# B&R Automation Studio project DuctLines (part 7)

#### Cyclic.ld
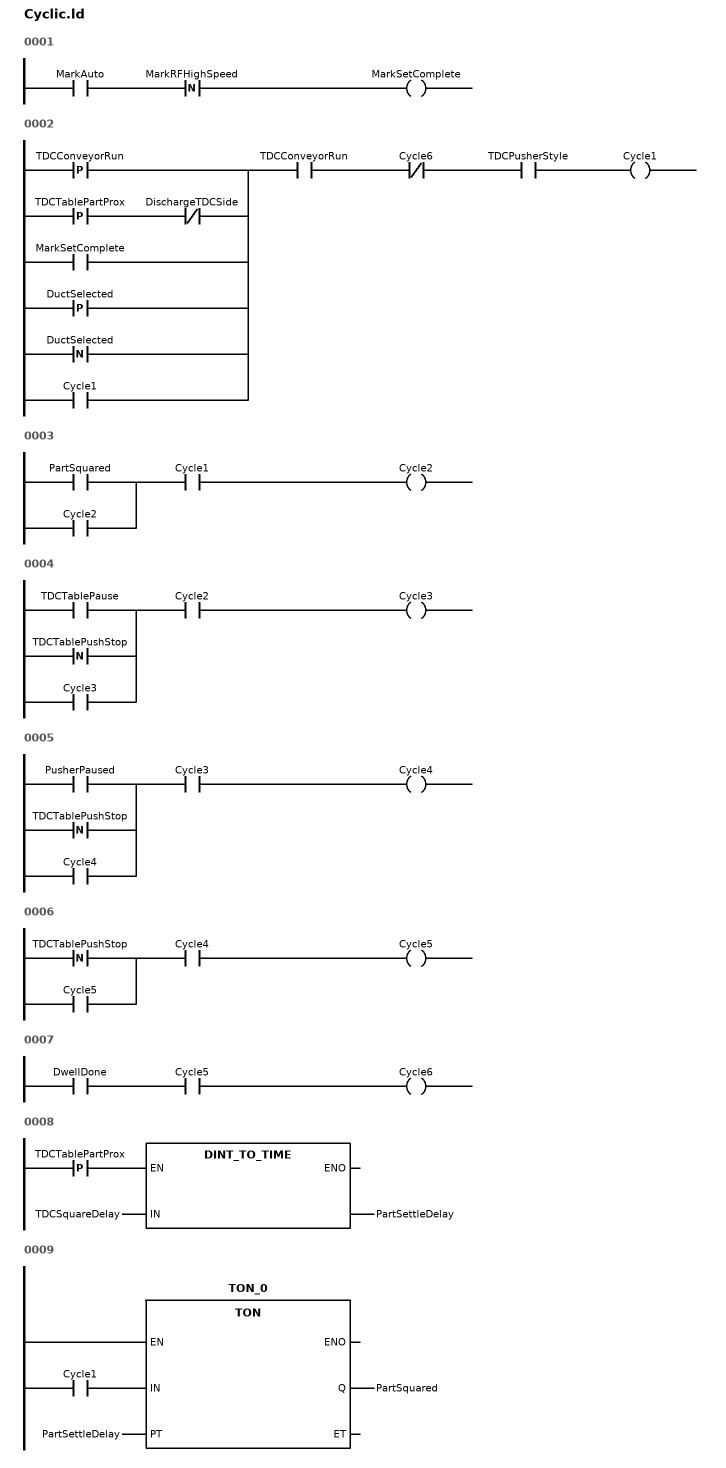
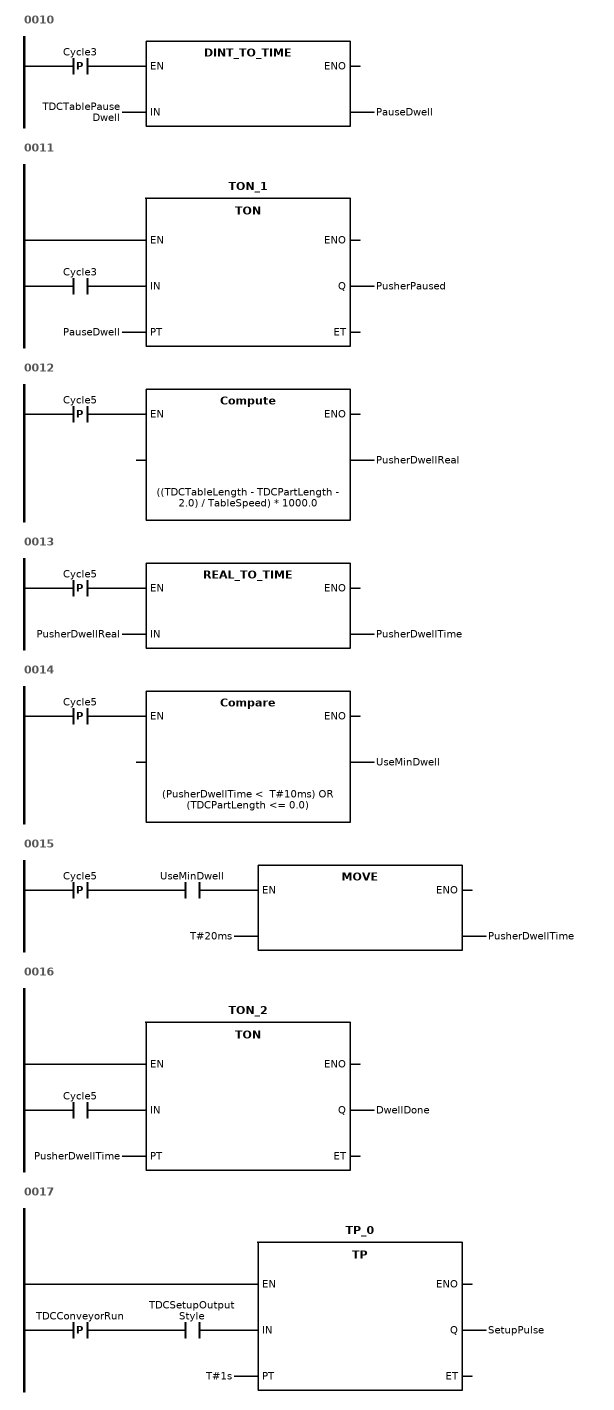
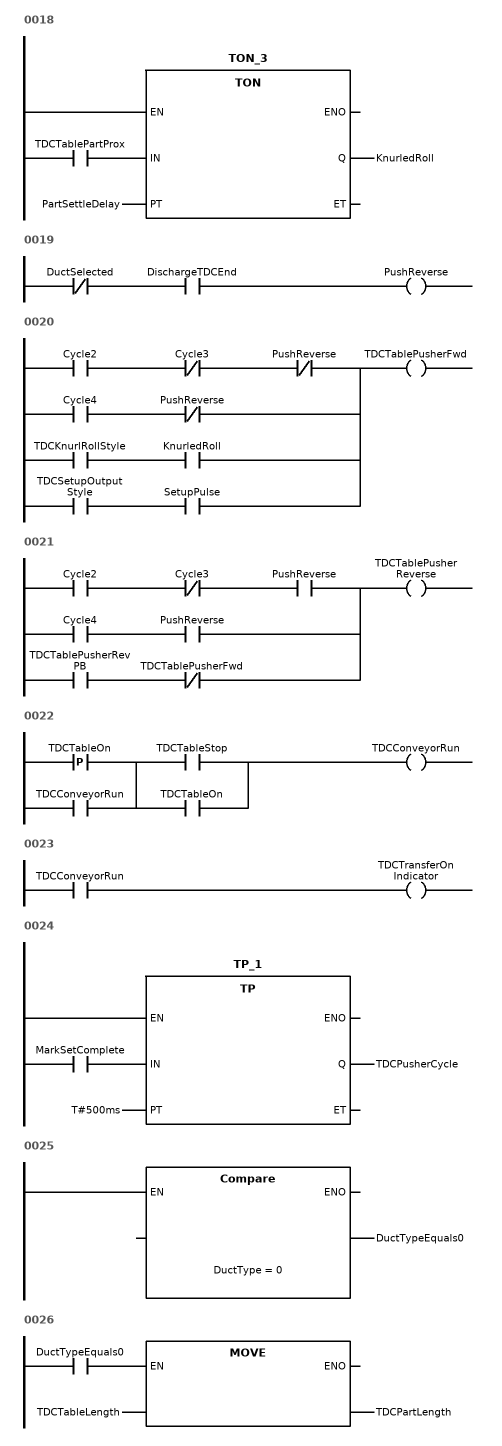
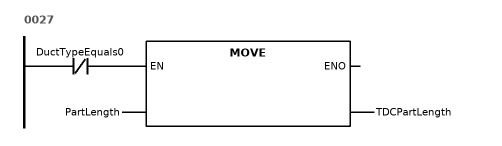
Ladder, written as Structured Text:
```iecst
PROGRAM _CYCLIC
VAR
    _e1 : F_TRIG;
    _e2 : R_TRIG;
    _e3 : R_TRIG;
    _e4 : R_TRIG;
    _e5 : F_TRIG;
    _e6 : F_TRIG;
    _e7 : F_TRIG;
    _e8 : F_TRIG;
    _e9 : R_TRIG;
    _e10 : R_TRIG;
    _e11 : R_TRIG;
    _e12 : R_TRIG;
    _e13 : R_TRIG;
    _e14 : R_TRIG;
    _e15 : R_TRIG;
    _e16 : R_TRIG;
END_VAR
(* Network 1 *)
_e1(CLK := MarkRFHighSpeed);
MarkSetComplete := MarkAuto AND _e1.Q;

(* Network 2 *)
_e2(CLK := TDCConveyorRun);
_e3(CLK := TDCTablePartProx);
_e4(CLK := DuctSelected);
_e5(CLK := DuctSelected);
Cycle1 := (_e2.Q OR (_e3.Q AND NOT DischargeTDCSide) OR MarkSetComplete OR _e4.Q OR _e5.Q OR Cycle1) AND TDCConveyorRun AND NOT Cycle6 AND TDCPusherStyle;

(* Network 3 *)
Cycle2 := (PartSquared OR Cycle2) AND Cycle1;

(* Network 4 *)
_e6(CLK := TDCTablePushStop);
Cycle3 := (TDCTablePause OR _e6.Q OR Cycle3) AND Cycle2;

(* Network 5 *)
_e7(CLK := TDCTablePushStop);
Cycle4 := (PusherPaused OR _e7.Q OR Cycle4) AND Cycle3;

(* Network 6 *)
_e8(CLK := TDCTablePushStop);
Cycle5 := (_e8.Q OR Cycle5) AND Cycle4;

(* Network 7 *)
Cycle6 := DwellDone AND Cycle5;

(* Network 8 *)
_e9(CLK := TDCTablePartProx);
IF _e9.Q THEN PartSettleDelay := DINT_TO_TIME(TDCSquareDelay); END_IF;

(* Network 9 *)
TON_0(IN := Cycle1, PT := PartSettleDelay);
PartSquared := TON_0.Q;

(* Network 10 *)
_e10(CLK := Cycle3);
IF _e10.Q THEN PauseDwell := DINT_TO_TIME(TDCTablePauseDwell); END_IF;

(* Network 11 *)
TON_1(IN := Cycle3, PT := PauseDwell);
PusherPaused := TON_1.Q;

(* Network 12 *)
_e11(CLK := Cycle5);
IF _e11.Q THEN PusherDwellReal := ((TDCTableLength - TDCPartLength - 2.0) / TableSpeed) * 1000.0; END_IF;

(* Network 13 *)
_e12(CLK := Cycle5);
IF _e12.Q THEN PusherDwellTime := REAL_TO_TIME(PusherDwellReal); END_IF;

(* Network 14 *)
_e13(CLK := Cycle5);
IF _e13.Q THEN UseMinDwell := (PusherDwellTime <  T#10ms) OR (TDCPartLength <= 0.0); END_IF;

(* Network 15 *)
_e14(CLK := Cycle5);
IF _e14.Q AND UseMinDwell THEN PusherDwellTime := T#20ms; END_IF;

(* Network 16 *)
TON_2(IN := Cycle5, PT := PusherDwellTime);
DwellDone := TON_2.Q;

(* Network 17 *)
_e15(CLK := TDCConveyorRun);
TP_0(IN := _e15.Q AND TDCSetupOutputStyle, PT := T#1s);
SetupPulse := TP_0.Q;

(* Network 18 *)
TON_3(IN := TDCTablePartProx, PT := PartSettleDelay);
KnurledRoll := TON_3.Q;

(* Network 19 *)
PushReverse := NOT DuctSelected AND DischargeTDCEnd;

(* Network 20 *)
TDCTablePusherFwd := (Cycle2 AND NOT Cycle3 AND NOT PushReverse) OR (Cycle4 AND NOT PushReverse) OR (TDCKnurlRollStyle AND KnurledRoll) OR (TDCSetupOutputStyle AND SetupPulse);

(* Network 21 *)
TDCTablePusherReverse := (Cycle2 AND NOT Cycle3 AND PushReverse) OR (Cycle4 AND PushReverse) OR (TDCTablePusherRevPB AND NOT TDCTablePusherFwd);

(* Network 22 *)
_e16(CLK := TDCTableOn);
TDCConveyorRun := (_e16.Q OR TDCConveyorRun) AND (TDCTableStop OR TDCTableOn);

(* Network 23 *)
TDCTransferOnIndicator := TDCConveyorRun;

(* Network 24 *)
TP_1(IN := MarkSetComplete, PT := T#500ms);
TDCPusherCycle := TP_1.Q;

(* Network 25 *)
DuctTypeEquals0 := DuctType = 0;

(* Network 26 *)
IF DuctTypeEquals0 THEN TDCPartLength := TDCTableLength; END_IF;

(* Network 27 *)
IF NOT DuctTypeEquals0 THEN TDCPartLength := PartLength; END_IF;
END_PROGRAM
```

### Program Logical/IMotionControl (IEC) - Ducto Roll Drive Electric Servo routine

#### Cyclic.st
```iecst
PROGRAM _CYCLIC
	difference := MetalTarget - ActlMetalEncoder;
	AbsoluteDifference := ABS(difference);
	CASE MotionStatus1 OF
		(*Hold Position*)
		0:
			IF NOT InPosition1 THEN
				IF AbsoluteDifference <= MetalTolerance THEN
					TargetCount1 := TargetCount1 + UpdateRate2;
					IF TargetCount1 >= SettleTime1 THEN
						InPosition1 := TRUE;
					END_IF;
				END_IF;
			END_IF;

			(*Ratio1 := DINT_TO_INT(difference + (difference / 1));*)
			Ratio1 := DINT_TO_INT(difference * 15);
			IF Counter1 > 0 THEN
				Counter1 := Counter1 - UpdateRate1;
			ELSE
				Counter1 := 500;
				IF Hold1 <> Ratio1 THEN
					Hold1 := Ratio1;
				ELSE
					DACBalance1 := ActualDAC1;
				END_IF;
			END_IF;

	    	TargetDAC1 := Ratio1 + DACBalance1;
			ActualDAC1 := TargetDAC1;
		(*	IF TargetDAC1 >= ActualDAC1 THEN
				IF TargetDAC1 - ActualDAC1 > (10 * UpdateRate1) THEN
					ActualDAC1 := ActualDAC1 + (10 * UpdateRate1);
				ELSE
					ActualDAC1 := TargetDAC1;
				END_IF;
			ELSE
				IF ActualDAC1 - TargetDAC1 > (10 * UpdateRate1) THEN
					ActualDAC1 := ActualDAC1 - (10 * UpdateRate1);
				ELSE
					ActualDAC1 := TargetDAC1;
				END_IF;
			END_IF;*)

			IF ActualDAC1 > TopDAC1 THEN
				ActualDAC1 := TopDAC1;
			END_IF;
			IF ActualDAC1 < -TopDAC1 THEN
				ActualDAC1 := -TopDAC1;
			END_IF

		(*Initialize Move*)
		1:
			CoilAccumulator := MetalTarget; (*Update Accumulator to last target*)
			(*IncrementalRealTarget is the amount required to move determined elsewhere*)
			IncrementalDINTTarget := REAL_TO_DINT(IncrementalRealTarget * UnitsPerInch1 * MetalScaler);
			MetalTarget := MetalTarget + IncrementalDINTTarget;
			DACAdd1 := INT_TO_REAL(MaxDAC) / AccelRampReal;
			ActualSpeed1 := (TopLineSpeed * DINT_TO_REAL(RunSpeed1)) / 100.0; (*Real Inches Per Second*)
			ActualRunPercent := ActualSpeed1 / (MaxSpeed1 / 5.0);
			IF ActualRunPercent > 1.0 THEN
				ActualRunPercent := 1.0;
			END_IF;
			TopDAC1 := REAL_TO_INT(INT_TO_REAL(MaxDAC) * ActualRunPercent);
			IF ActualRunPercent = 1.0 THEN
				TopDAC1 := TopDAC1 - REAL_TO_INT(DACAdd1);
			END_IF;

			AverageSpeed1 := ActualSpeed1 / 2.0;
			DecelTime1 := (DecelRampReal / 1000.0) * ActualRunPercent;
			DecelDistance1 := REAL_TO_DINT(((AverageSpeed1 * DecelTime1 ) * MetalScaler) * UnitsPerInch1);
			MaxCountsPerSecond := (MaxSpeed1 / 5.0) * UnitsPerInch1;
			SRM1 := MaxDACSquared / ((MaxCountsPerSecond * (DecelRampReal / 1000.0)) / 2.0);
			(*SRM1 := MaxDACSquared / ((MaxCountsPerSecond * (DecelRampReal / 1000.0)));*)
			IF DecelDistance1 > (IncrementalDINTTarget / 2) THEN
				DecelDistance1 := IncrementalDINTTarget / 2;
				TopDAC1 := REAL_TO_INT(SQRT((DINT_TO_REAL(DecelDistance1) / MetalScaler) * SRM1));
				IF TopDAC1 < 3276 THEN
					TopDAC1 := 3276;
				END_IF;
			END_IF;
			InPosition1 := FALSE;
			FirstTarget1 := FALSE;
			StopWatch1 := 0.0;
			MotionStatus1 := 2;
		(*Ramp Up To Speed*)
		2:
			IF DecelDistance1 < difference THEN
				IF ActualDAC1 < TopDAC1 THEN (*Accelerate*)
					StopWatch1 := StopWatch1 + INT_TO_REAL(UpdateRate1);
					ActualDAC1 := REAL_TO_INT(StopWatch1 * DACAdd1);
				ELSE  (*Constant Speed*)
					ActualDAC1 := TopDAC1;
				END_IF;
			ELSE (*Switch To Decel MotionState*)
				DecelCounter := 25;
				LastPosition1 := ActlMetalEncoder;
				TargetCount1 := 0;
				FirstTarget1 := FALSE	;
				MotionStatus1 := 3;
			END_IF;
		3:
			(*Stall Detection*)
			DecelCounter := DecelCounter - UpdateRate1;
			IF DecelCounter <= 0 THEN
				DecelCounter := 200;
				IF LastPosition1 = ActlMetalEncoder THEN
					DACBalance1 := ActualDAC1;
					Counter1 := 0;
					TopDAC1 := MaxDAC / 4;
					MotionStatus1 := 0;
				ELSE
					LastPosition1 := ActlMetalEncoder;
				END_IF;
			END_IF;

			RealDAC1 := REAL_TO_INT(SQRT(DINT_TO_REAL(AbsoluteDifference) * SRM1));
			IF RealDAC1 > INT_TO_REAL(MaxDAC) THEN
				RealDAC1 := INT_TO_REAL(MaxDAC);
			END_IF;
			ActualDAC1 := REAL_TO_INT(RealDAC1);

			IF difference < 0 THEN
				ActualDAC1 := -ActualDAC1;
			END_IF;

			IF FirstTarget1 THEN
				ActualDAC1 := ActualDAC1 / 8;
			END_IF;

			IF AbsoluteDifference < MetalTolerance THEN
				FirstTarget1 := TRUE;
				TargetCount1 := TargetCount1 + UpdateRate1;
				IF TargetCount1 >= SettleTime1 THEN
					Counter1 := 0;
					InPosition1 := TRUE;
					MotionStatus1 := 0;
					TopDAC1 := MaxDAC / 4;
				END_IF;
			ELSE
				TargetCount1 := 0;
			END_IF;
		4: (*Setup Forward Jog*)
			DACAdd1 := INT_TO_REAL(MaxDAC) / AccelRampReal;
			TopDAC1 := DINT_TO_INT((INT_TO_DINT(MaxDAC) * PercentJogSpeed1) / 100);
			TopDAC1 := TopDAC1 - REAL_TO_INT(DACAdd1);
			StopFlag1 := FALSE;
			MotionStatus1 := 7;
		5: (*Setup Reverse Jog*)
			DACAdd1 := INT_TO_REAL(MaxDAC) / AccelRampReal;
			TopDAC1 := DINT_TO_INT((INT_TO_DINT(MaxDAC) * PercentJogSpeed1) / 100);
			TopDAC1 := TopDAC1 - REAL_TO_INT(DACAdd1);
			StopFlag1 := FALSE;
			MotionStatus1 := 8;
		7: (*Forward Jog*)
			IF StopFlag1 THEN
				IF ActualDAC1 > REAL_TO_INT(DACAdd1) THEN (*Decelerate*)
					ActualDAC1 := ActualDAC1 - REAL_TO_INT(DACAdd1);
				ELSE (*Hold Position*)
					ActualDAC1 := 0;
					MetalTarget := ActlMetalEncoder;
					InPosition1 := TRUE;
					MotionStatus1 := -1;
				END_IF;
			ELSE
				InPosition1 := FALSE;
				IF ActualDAC1 < TopDAC1 THEN (*Accelerate*)
					ActualDAC1 := ActualDAC1 + REAL_TO_INT(DACAdd1);
				ELSE
					ActualDAC1 := TopDAC1; (*Maintain Constant Speed*)
				END_IF;
			END_IF;
		8: (*Reverse Jog*)
			IF StopFlag1 THEN
				IF ActualDAC1 < REAL_TO_INT(-DACAdd1) THEN (*Decelerate*)
					ActualDAC1 := ActualDAC1 + REAL_TO_INT(DACAdd1);
				ELSE (*Hold Position*)
					ActualDAC1 := 0;
					MetalTarget := ActlMetalEncoder;
					InPosition1 := TRUE;
					MotionStatus1 := -1;
				END_IF;
			ELSE
				(*Don't Do This To Prevent Uncoiler From Running Forward*)
				(*InPosition1 := FALSE;*)
				IF ActualDAC1 > -TopDAC1 THEN (*Accelerate*)
					ActualDAC1 := ActualDAC1 - REAL_TO_INT(DACAdd1);
				ELSE
					ActualDAC1 := -TopDAC1; (*Maintain Constant Speed*)
				END_IF;
			END_IF;
		9:
			IF ActualDAC1 > REAL_TO_INT(DACAdd1) THEN (*Decelerate*)
				ActualDAC1 := ActualDAC1 - REAL_TO_INT(DACAdd1);
			ELSE (* Hold Position *)
				MetalTarget := ActlMetalEncoder;
				IncrementalRealTarget := DINT_TO_REAL(difference) / UnitsPerInch1 / MetalScaler;
				MotionStatus1 := 0;
			END_IF;
		ELSE (*Not Moving Or Holding*)
		  ActualDAC1 := 0;
		  MetalTarget := ActlMetalEncoder;
		  InPosition1 := TRUE;
	END_CASE;

	IF ActualDAC1 > MaxDAC THEN
		ActualDAC1 := MaxDAC;
	END_IF;
	IF ActualDAC1 < -MaxDAC THEN
		ActualDAC1 := -MaxDAC;
	END_IF;

END_PROGRAM
```

### Program Logical/HydraulicBrakeCarriage (IEC) - Reference Sequence for all brakes begins around rung #9, Move To Target Logic For Digital Output controlled brakes begins rung #15, Wrap Brake With PLC Outputs about rung #48

#### Variables.var
```iecst
VAR
	AbsDifference : REAL;
	BSWReal : REAL;
	DecelDone1 : BOOL;
	DecelDone2 : BOOL;
	DifferenceGreaterThan0 : BOOL;
	InPosWindow : BOOL;
	InSSWindow : BOOL;
	LLimit : REAL;
	MCLessThan0 : BOOL;
	MinusStop : BOOL;
	Move4HWBwoPLC : BOOL;
	MoveMinus4 : BOOL;
	MovePlus4 : BOOL;
	MVMinusUnlatch : BOOL;
	MVPlusUnlatch : BOOL;
	PlusStop : BOOL;
	PositioningError1 : BOOL;
	PositioningError2 : BOOL;
	realBTW : REAL;
	ROffSignal : BOOL;
	SettleTime : TIME := T#1500ms;
	SSWin : REAL;
	TON_1 : TON;
	TON_2 : TON;
	TON_3 : TON;
	TON_4 : TON;
	TON_5 : TON;
	ULimit : REAL;
	TON_0 : TON;
	HWBwPLC_H7 : BOOL;
	BC_Home1 : BOOL;
	BC_Home2 : BOOL;
	BC_Home3 : BOOL;
	TON_6 : TON;
	BPositionUpdateDelayDone : BOOL;
	TON_7 : TON;
	CarriagePositionUpdateDwell : BOOL;
	BC_Home5 : BOOL;
	BCForwardTravelLimit : BOOL;
	BCReverseTravelLimit : BOOL;
	SetLBrakeCarriage : BOOL;
	HWBrakeHomed : BOOL;
	HoldingPosition : BOOL;
	BC_Home2B : BOOL;
	TempBrakeCarriageTarget : REAL;
	FirstCycle : BOOL;
	TP_0 : TP;
	BCTLessThan0 : BOOL;
END_VAR
```

#### Cyclic.ld
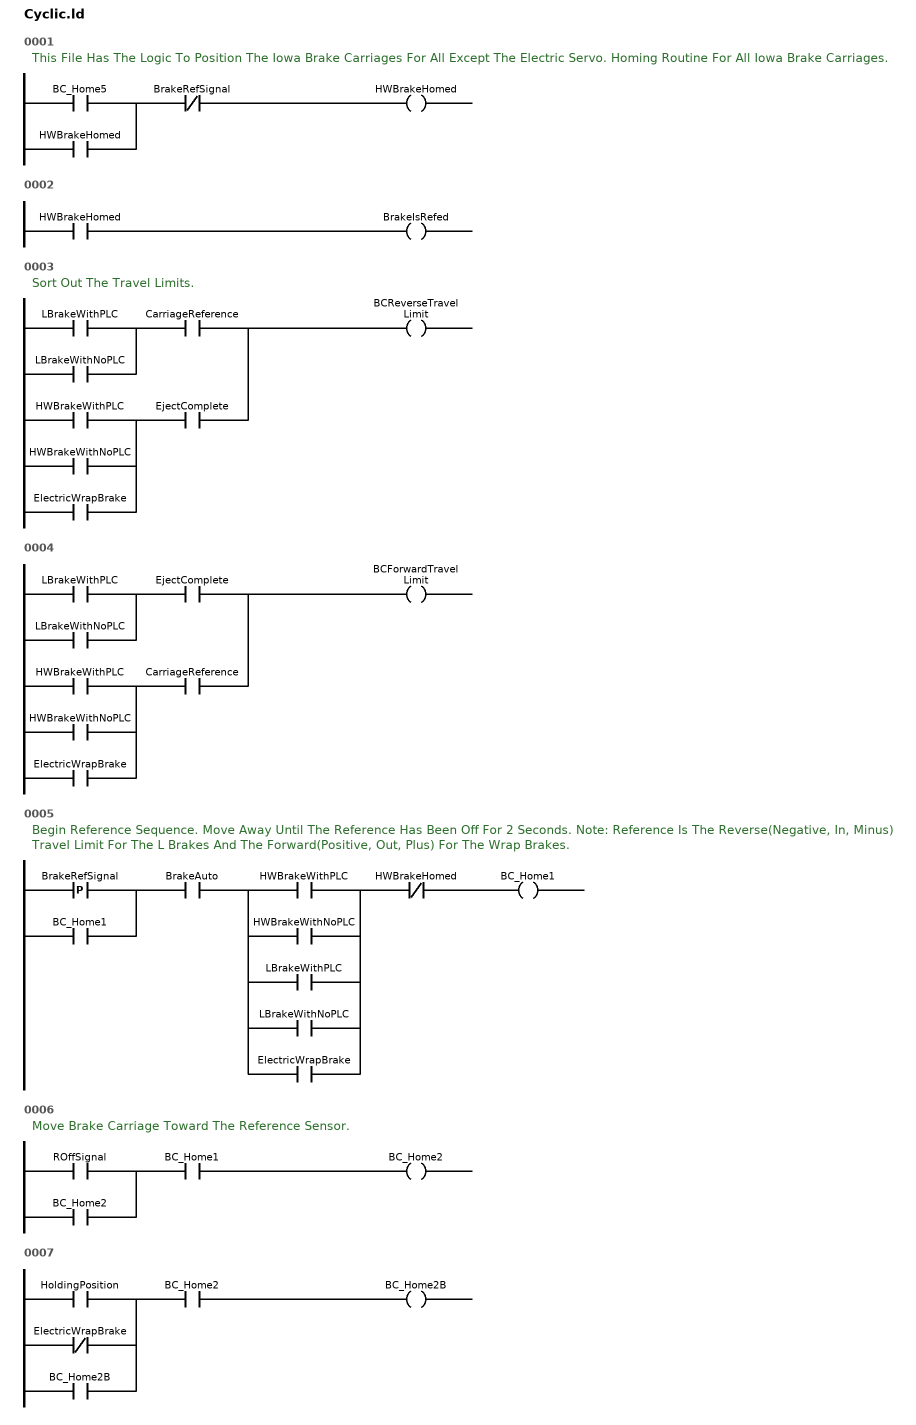
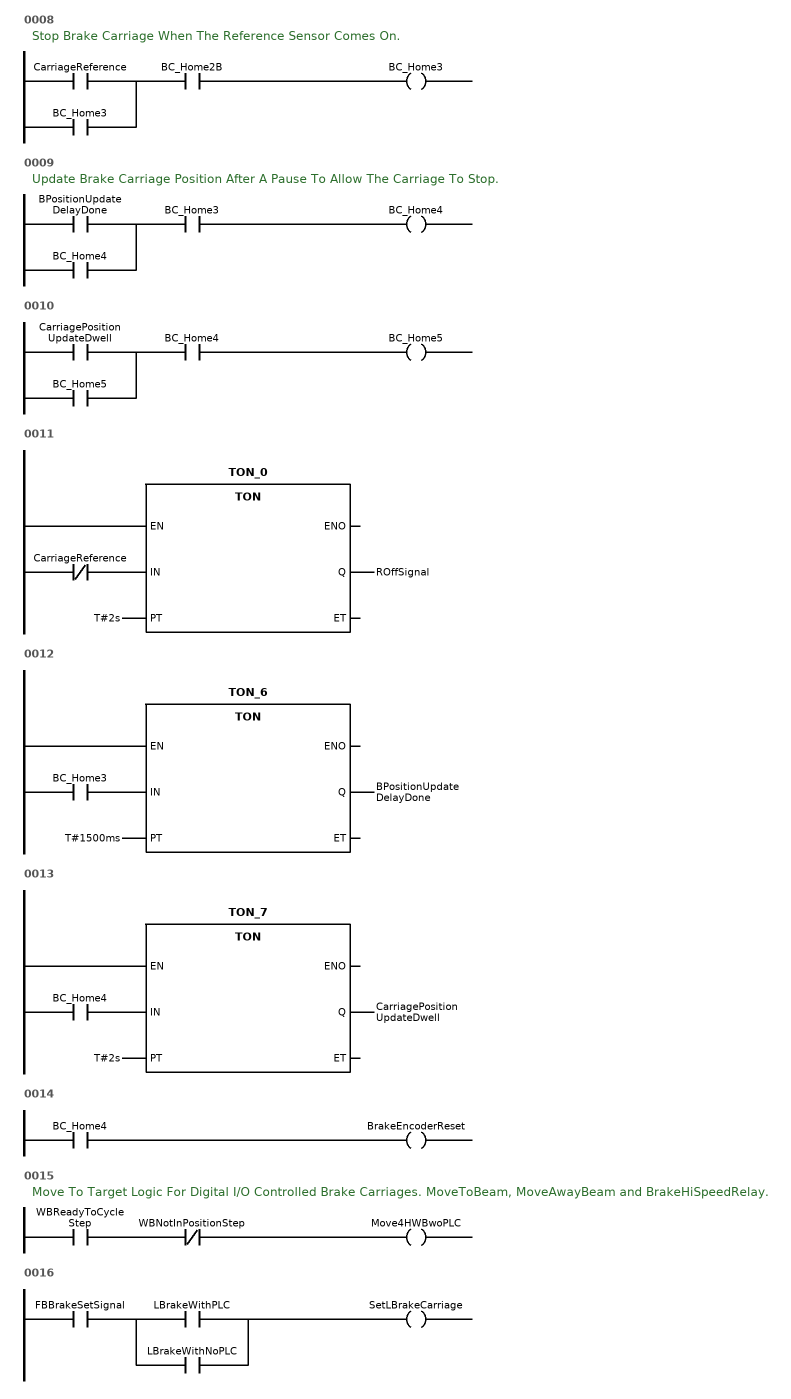
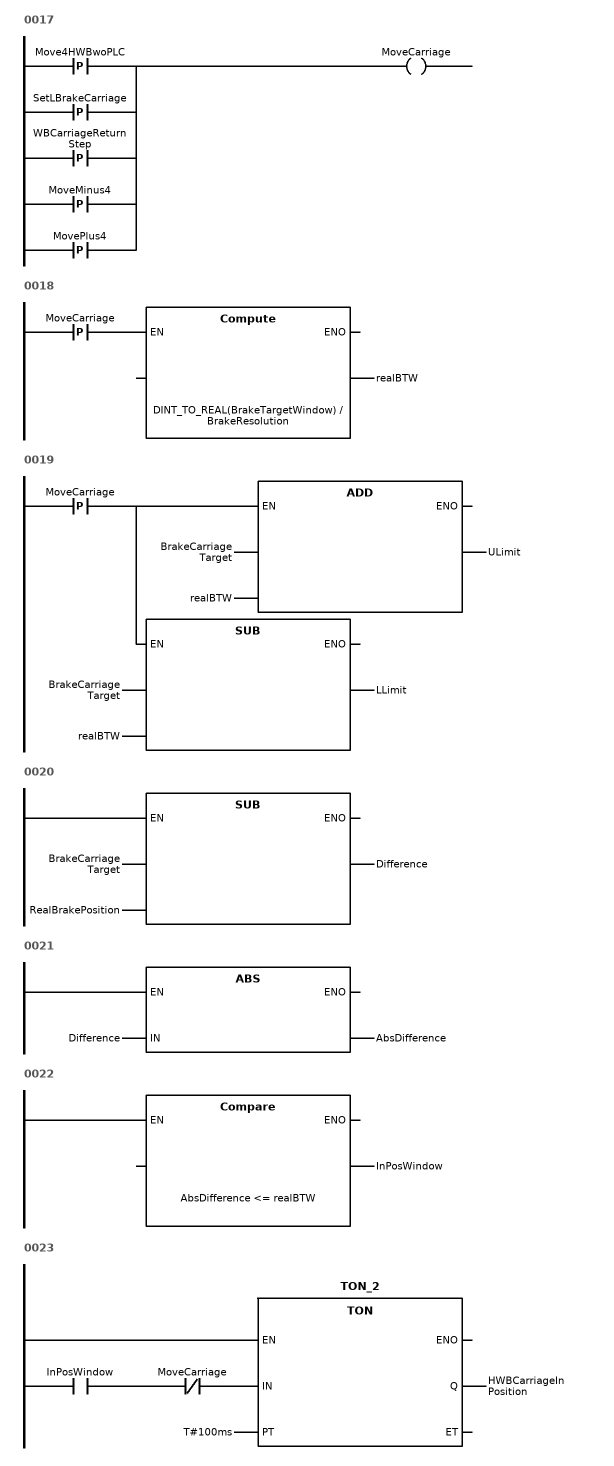
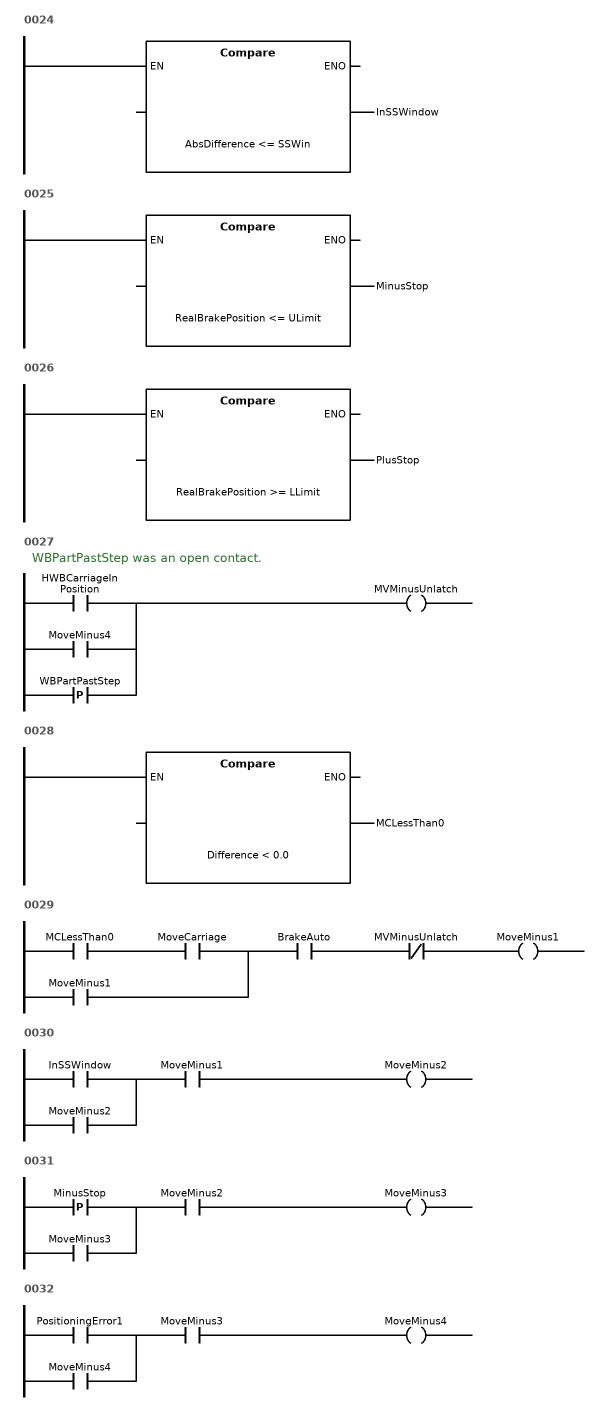
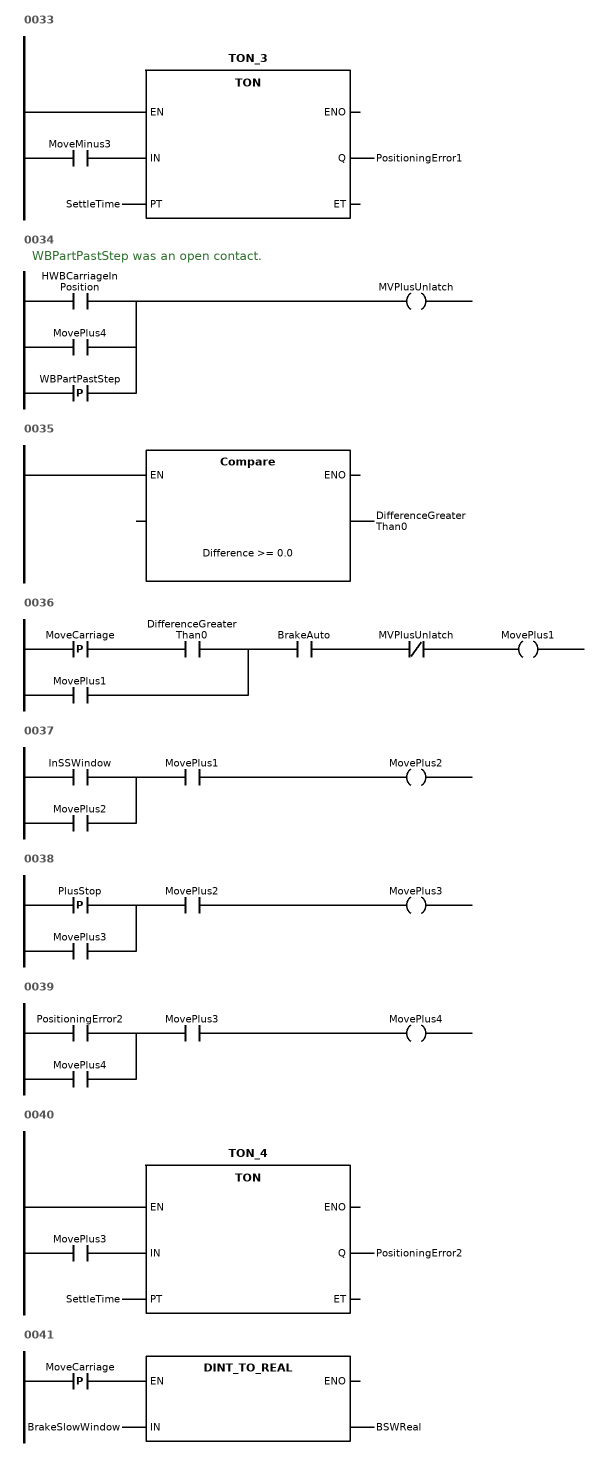
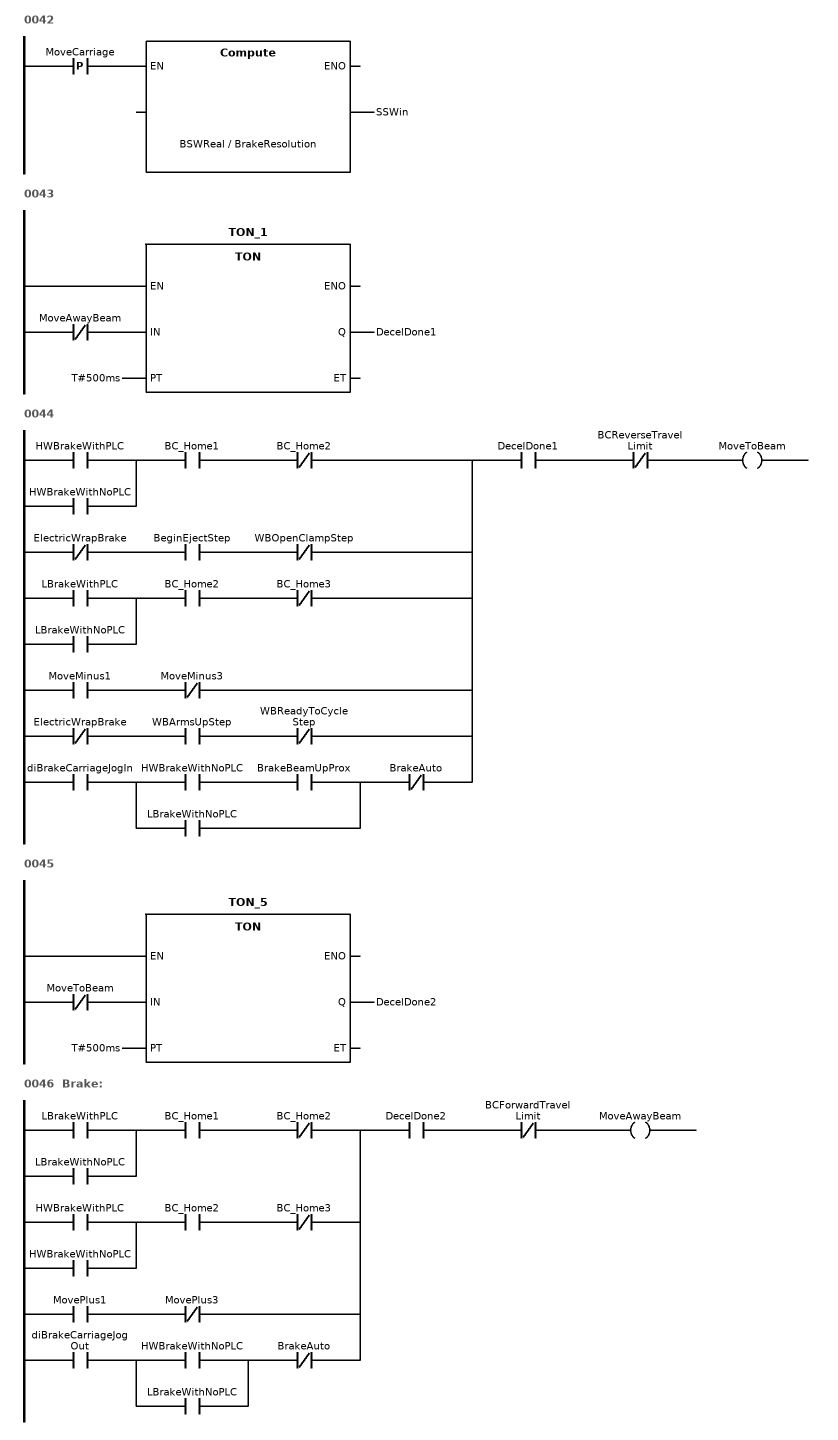
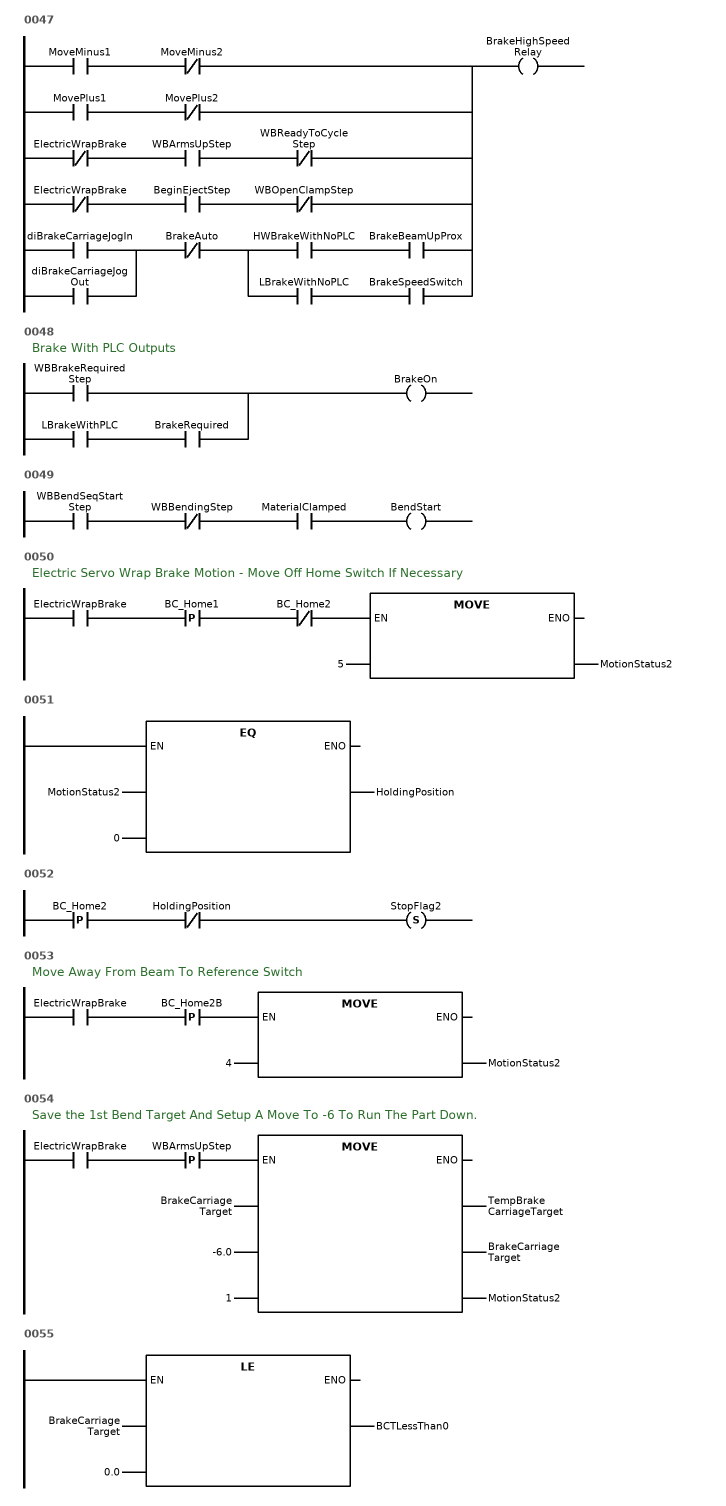
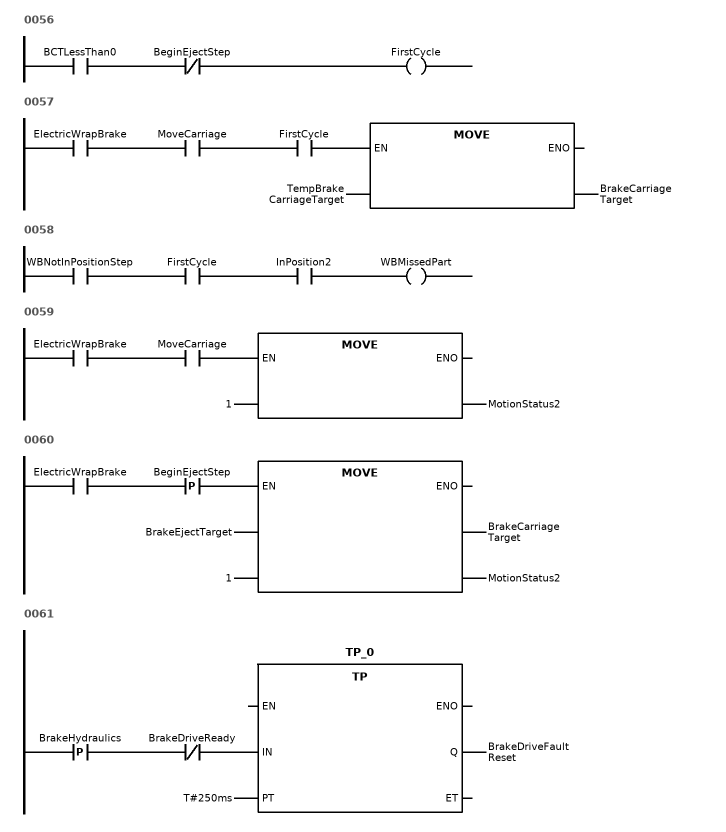
Ladder, written as Structured Text:
```iecst
PROGRAM _CYCLIC
VAR
    _e1 : R_TRIG;
    _e2 : R_TRIG;
    _e3 : R_TRIG;
    _e4 : R_TRIG;
    _e5 : R_TRIG;
    _e6 : R_TRIG;
    _e7 : R_TRIG;
    _e8 : R_TRIG;
    _e9 : R_TRIG;
    _e10 : R_TRIG;
    _e11 : R_TRIG;
    _e12 : R_TRIG;
    _e13 : R_TRIG;
    _e14 : R_TRIG;
    _e15 : R_TRIG;
    _p16 : BOOL;
    _e17 : R_TRIG;
    _e18 : R_TRIG;
    _e19 : R_TRIG;
    _e20 : R_TRIG;
    _e21 : R_TRIG;
    _e22 : R_TRIG;
END_VAR
(* Network 1: This File Has The Logic To Position The Iowa Brake Carriages For All Except The Electric Servo. Homing Routine For All Iowa Brake Carriages. *)
HWBrakeHomed := (BC_Home5 OR HWBrakeHomed) AND NOT BrakeRefSignal;

(* Network 2 *)
BrakeIsRefed := HWBrakeHomed;

(* Network 3: Sort Out The Travel Limits. *)
BCReverseTravelLimit := ((LBrakeWithPLC OR LBrakeWithNoPLC) AND CarriageReference) OR ((HWBrakeWithPLC OR HWBrakeWithNoPLC OR ElectricWrapBrake) AND EjectComplete);

(* Network 4 *)
BCForwardTravelLimit := ((LBrakeWithPLC OR LBrakeWithNoPLC) AND EjectComplete) OR ((HWBrakeWithPLC OR HWBrakeWithNoPLC OR ElectricWrapBrake) AND CarriageReference);

(* Network 5: Begin Reference Sequence. Move Away Until The Reference Has Been Off For 2 Seconds. Note: Reference Is The Reverse(Negative, In, Minus) Travel Limit For The L Brakes And The Forward(Positive, Out, Plus) For The Wrap Brakes.  *)
_e1(CLK := BrakeRefSignal);
BC_Home1 := (_e1.Q OR BC_Home1) AND BrakeAuto AND (HWBrakeWithPLC OR HWBrakeWithNoPLC OR LBrakeWithPLC OR LBrakeWithNoPLC OR ElectricWrapBrake) AND NOT HWBrakeHomed;

(* Network 6: Move Brake Carriage Toward The Reference Sensor. *)
BC_Home2 := (ROffSignal OR BC_Home2) AND BC_Home1;

(* Network 7 *)
BC_Home2B := (HoldingPosition OR NOT ElectricWrapBrake OR BC_Home2B) AND BC_Home2;

(* Network 8: Stop Brake Carriage When The Reference Sensor Comes On. *)
BC_Home3 := (CarriageReference OR BC_Home3) AND BC_Home2B;

(* Network 9: Update Brake Carriage Position After A Pause To Allow The Carriage To Stop. *)
BC_Home4 := (BPositionUpdateDelayDone OR BC_Home4) AND BC_Home3;

(* Network 10 *)
BC_Home5 := (CarriagePositionUpdateDwell OR BC_Home5) AND BC_Home4;

(* Network 11 *)
TON_0(IN := NOT CarriageReference, PT := T#2s);
ROffSignal := TON_0.Q;

(* Network 12 *)
TON_6(IN := BC_Home3, PT := T#1500ms);
BPositionUpdateDelayDone := TON_6.Q;

(* Network 13 *)
TON_7(IN := BC_Home4, PT := T#2s);
CarriagePositionUpdateDwell := TON_7.Q;

(* Network 14 *)
BrakeEncoderReset := BC_Home4;

(* Network 15: Move To Target Logic For Digital I/O Controlled Brake Carriages. MoveToBeam, MoveAwayBeam and BrakeHiSpeedRelay. *)
Move4HWBwoPLC := WBReadyToCycleStep AND NOT WBNotInPositionStep;

(* Network 16 *)
SetLBrakeCarriage := FBBrakeSetSignal AND (LBrakeWithPLC OR LBrakeWithNoPLC);

(* Network 17 *)
_e2(CLK := Move4HWBwoPLC);
_e3(CLK := SetLBrakeCarriage);
_e4(CLK := WBCarriageReturnStep);
_e5(CLK := MoveMinus4);
_e6(CLK := MovePlus4);
MoveCarriage := _e2.Q OR _e3.Q OR _e4.Q OR _e5.Q OR _e6.Q;

(* Network 18 *)
_e7(CLK := MoveCarriage);
IF _e7.Q THEN realBTW := DINT_TO_REAL(BrakeTargetWindow) / BrakeResolution; END_IF;

(* Network 19 *)
_e8(CLK := MoveCarriage);
IF _e8.Q THEN
    ULimit := BrakeCarriageTarget + realBTW;
    LLimit := BrakeCarriageTarget - realBTW;
END_IF;

(* Network 20 *)
Difference := BrakeCarriageTarget - RealBrakePosition;

(* Network 21 *)
AbsDifference := ABS(Difference);

(* Network 22 *)
InPosWindow := AbsDifference <= realBTW;

(* Network 23 *)
TON_2(IN := InPosWindow AND NOT MoveCarriage, PT := T#100ms);
HWBCarriageInPosition := TON_2.Q;

(* Network 24 *)
InSSWindow := AbsDifference <= SSWin;

(* Network 25 *)
MinusStop := RealBrakePosition <= ULimit;

(* Network 26 *)
PlusStop := RealBrakePosition >= LLimit;

(* Network 27: WBPartPastStep was an open contact. *)
_e9(CLK := WBPartPastStep);
MVMinusUnlatch := HWBCarriageInPosition OR MoveMinus4 OR _e9.Q;

(* Network 28 *)
MCLessThan0 := Difference < 0.0;

(* Network 29 *)
MoveMinus1 := ((MCLessThan0 AND MoveCarriage) OR MoveMinus1) AND BrakeAuto AND NOT MVMinusUnlatch;

(* Network 30 *)
MoveMinus2 := (InSSWindow OR MoveMinus2) AND MoveMinus1;

(* Network 31 *)
_e10(CLK := MinusStop);
MoveMinus3 := (_e10.Q OR MoveMinus3) AND MoveMinus2;

(* Network 32 *)
MoveMinus4 := (PositioningError1 OR MoveMinus4) AND MoveMinus3;

(* Network 33 *)
TON_3(IN := MoveMinus3, PT := SettleTime);
PositioningError1 := TON_3.Q;

(* Network 34: WBPartPastStep was an open contact. *)
_e11(CLK := WBPartPastStep);
MVPlusUnlatch := HWBCarriageInPosition OR MovePlus4 OR _e11.Q;

(* Network 35 *)
DifferenceGreaterThan0 := Difference >= 0.0;

(* Network 36 *)
_e12(CLK := MoveCarriage);
MovePlus1 := ((_e12.Q AND DifferenceGreaterThan0) OR MovePlus1) AND BrakeAuto AND NOT MVPlusUnlatch;

(* Network 37 *)
MovePlus2 := (InSSWindow OR MovePlus2) AND MovePlus1;

(* Network 38 *)
_e13(CLK := PlusStop);
MovePlus3 := (_e13.Q OR MovePlus3) AND MovePlus2;

(* Network 39 *)
MovePlus4 := (PositioningError2 OR MovePlus4) AND MovePlus3;

(* Network 40 *)
TON_4(IN := MovePlus3, PT := SettleTime);
PositioningError2 := TON_4.Q;

(* Network 41 *)
_e14(CLK := MoveCarriage);
IF _e14.Q THEN BSWReal := DINT_TO_REAL(BrakeSlowWindow); END_IF;

(* Network 42 *)
_e15(CLK := MoveCarriage);
IF _e15.Q THEN SSWin := BSWReal / BrakeResolution; END_IF;

(* Network 43 *)
TON_1(IN := NOT MoveAwayBeam, PT := T#500ms);
DecelDone1 := TON_1.Q;

(* Network 44 *)
MoveToBeam := (((HWBrakeWithPLC OR HWBrakeWithNoPLC) AND BC_Home1 AND NOT BC_Home2) OR (NOT ElectricWrapBrake AND BeginEjectStep AND NOT WBOpenClampStep) OR ((LBrakeWithPLC OR LBrakeWithNoPLC) AND BC_Home2 AND NOT BC_Home3) OR (MoveMinus1 AND NOT MoveMinus3) OR (NOT ElectricWrapBrake AND WBArmsUpStep AND NOT WBReadyToCycleStep) OR (diBrakeCarriageJogIn AND ((HWBrakeWithNoPLC AND BrakeBeamUpProx) OR LBrakeWithNoPLC) AND NOT BrakeAuto)) AND DecelDone1 AND NOT BCReverseTravelLimit;

(* Network 45 *)
TON_5(IN := NOT MoveToBeam, PT := T#500ms);
DecelDone2 := TON_5.Q;

(* Network 46 *)
Brake:
MoveAwayBeam := (((LBrakeWithPLC OR LBrakeWithNoPLC) AND BC_Home1 AND NOT BC_Home2) OR ((HWBrakeWithPLC OR HWBrakeWithNoPLC) AND BC_Home2 AND NOT BC_Home3) OR (MovePlus1 AND NOT MovePlus3) OR (diBrakeCarriageJogOut AND (HWBrakeWithNoPLC OR LBrakeWithNoPLC) AND NOT BrakeAuto)) AND DecelDone2 AND NOT BCForwardTravelLimit;

(* Network 47 *)
_p16 := (diBrakeCarriageJogIn OR diBrakeCarriageJogOut) AND NOT BrakeAuto;
BrakeHighSpeedRelay := (MoveMinus1 AND NOT MoveMinus2) OR (MovePlus1 AND NOT MovePlus2) OR (NOT ElectricWrapBrake AND ((WBArmsUpStep AND NOT WBReadyToCycleStep) OR (BeginEjectStep AND NOT WBOpenClampStep))) OR (_p16 AND ((HWBrakeWithNoPLC AND BrakeBeamUpProx) OR (LBrakeWithNoPLC AND BrakeSpeedSwitch)));

(* Network 48: Brake With PLC Outputs *)
BrakeOn := WBBrakeRequiredStep OR (LBrakeWithPLC AND BrakeRequired);

(* Network 49 *)
BendStart := WBBendSeqStartStep AND NOT WBBendingStep AND MaterialClamped;

(* Network 50: Electric Servo Wrap Brake Motion - Move Off Home Switch If Necessary *)
_e17(CLK := BC_Home1);
IF ElectricWrapBrake AND _e17.Q AND NOT BC_Home2 THEN MotionStatus2 := 5; END_IF;

(* Network 51 *)
HoldingPosition := MotionStatus2 = 0;

(* Network 52 *)
_e18(CLK := BC_Home2);
IF _e18.Q AND NOT HoldingPosition THEN StopFlag2 := TRUE; END_IF;

(* Network 53: Move Away From Beam To Reference Switch *)
_e19(CLK := BC_Home2B);
IF ElectricWrapBrake AND _e19.Q THEN MotionStatus2 := 4; END_IF;

(* Network 54: Save the 1st Bend Target And Setup A Move To -6 To Run The Part Down. *)
_e20(CLK := WBArmsUpStep);
IF ElectricWrapBrake AND _e20.Q THEN
    TempBrakeCarriageTarget := BrakeCarriageTarget;
    BrakeCarriageTarget := -6.0;
    MotionStatus2 := 1;
END_IF;

(* Network 55 *)
BCTLessThan0 := BrakeCarriageTarget <= 0.0;

(* Network 56 *)
FirstCycle := BCTLessThan0 AND NOT BeginEjectStep;

(* Network 57 *)
IF ElectricWrapBrake AND MoveCarriage AND FirstCycle THEN
    BrakeCarriageTarget := TempBrakeCarriageTarget;
END_IF;

(* Network 58 *)
WBMissedPart := WBNotInPositionStep AND FirstCycle AND InPosition2;

(* Network 59 *)
IF ElectricWrapBrake AND MoveCarriage THEN MotionStatus2 := 1; END_IF;

(* Network 60 *)
_e21(CLK := BeginEjectStep);
IF ElectricWrapBrake AND _e21.Q THEN
    BrakeCarriageTarget := BrakeEjectTarget;
    MotionStatus2 := 1;
END_IF;

(* Network 61 *)
_e22(CLK := BrakeHydraulics);
TP_0(IN := _e22.Q AND NOT BrakeDriveReady, PT := T#250ms);
BrakeDriveFaultReset := TP_0.Q;
END_PROGRAM
```

### Program Logical/CleatRoll (IEC)

#### Variables.var
```iecst
VAR
	tmCleatOnDelay : TIME;
	tmCleatOffDelay : TIME;
	CleatOff : DINT;
	Cleat1And3 : DINT;
	Cleat2And4 : DINT;
	CleatFull : DINT;
	CleatLeftSideOnly : DINT;
	CleatRightSideOnly : DINT;
	CleatBothSides : DINT;
	CleatLeft : BOOL;
	CleatRight : BOOL;
	CRReset : BOOL;
	cleat4 : BOOL;
	cleat1 : BOOL := FALSE;
	cleat2 : BOOL;
	cleat3 : BOOL;
	CleatOutput : BOOL;
	CleatOutputRaw : BOOL;
	TON_0 : TON;
	TOF_0 : TOF;
	CleatOutputDOB : BOOL;
	CleatOutputDOM : BOOL;
	TON_1 : TON;
	blCleat1And3 : BOOL;
	blCleat2And4 : BOOL;
	blCleatFull : BOOL;
END_VAR
```

#### Cyclic.ld
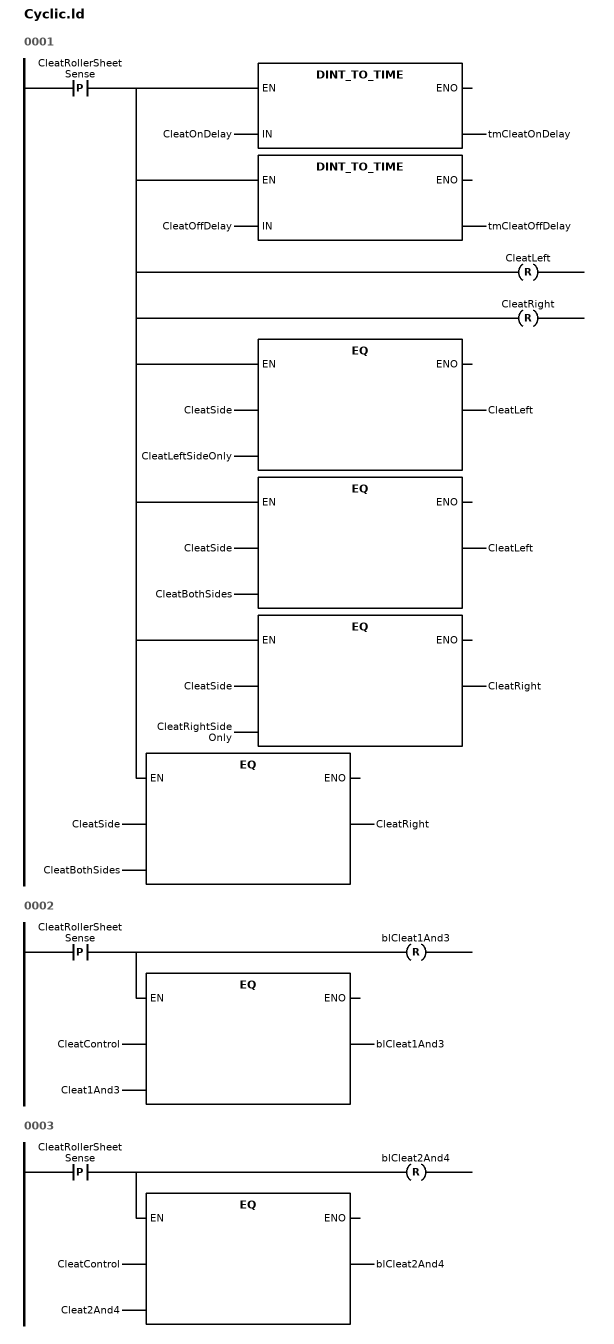
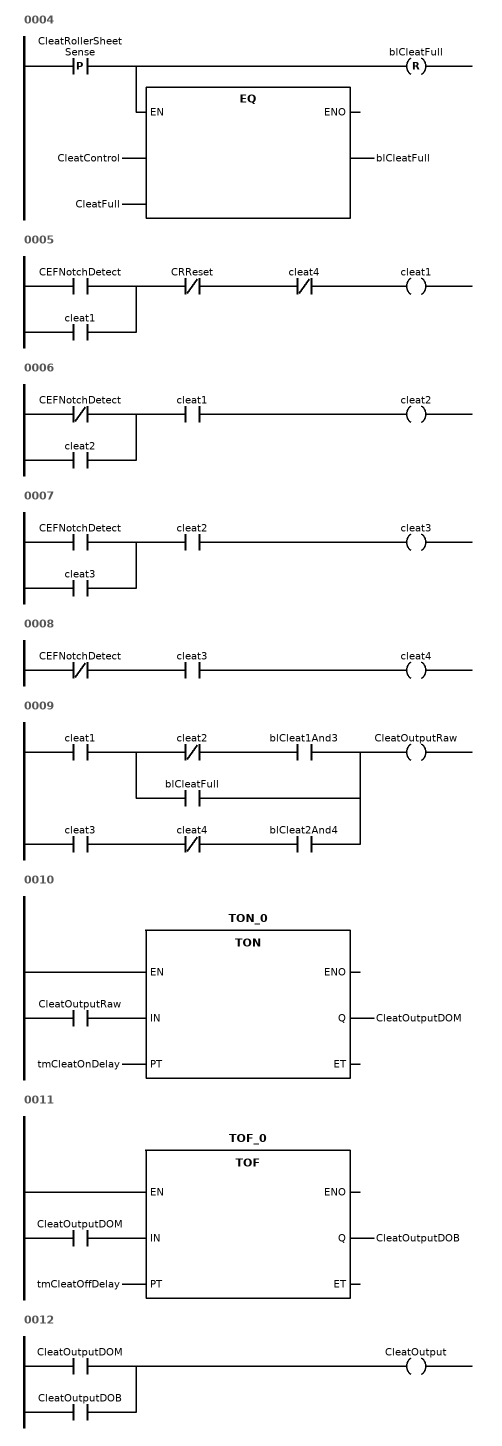
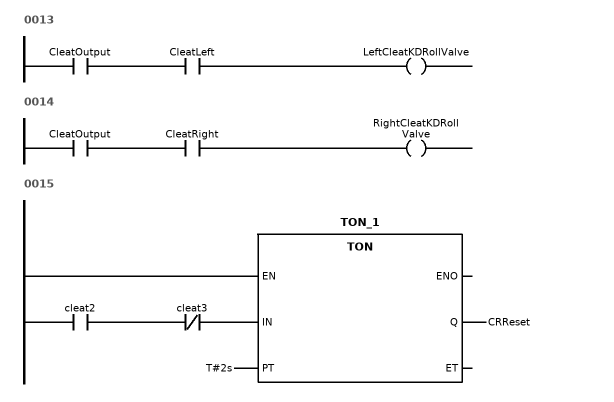
Ladder, written as Structured Text:
```iecst
PROGRAM _CYCLIC
VAR
    _e1 : R_TRIG;
    _e2 : R_TRIG;
    _e3 : R_TRIG;
    _e4 : R_TRIG;
END_VAR
(* Network 1 *)
_e1(CLK := CleatRollerSheetSense);
IF _e1.Q THEN
    tmCleatOnDelay := DINT_TO_TIME(CleatOnDelay);
    tmCleatOffDelay := DINT_TO_TIME(CleatOffDelay);
    CleatLeft := FALSE;
    CleatRight := FALSE;
    CleatLeft := CleatSide = CleatLeftSideOnly;
    CleatLeft := CleatSide = CleatBothSides;
    CleatRight := CleatSide = CleatRightSideOnly;
    CleatRight := CleatSide = CleatBothSides;
END_IF;

(* Network 2 *)
_e2(CLK := CleatRollerSheetSense);
IF _e2.Q THEN
    blCleat1And3 := FALSE;
    blCleat1And3 := CleatControl = Cleat1And3;
END_IF;

(* Network 3 *)
_e3(CLK := CleatRollerSheetSense);
IF _e3.Q THEN
    blCleat2And4 := FALSE;
    blCleat2And4 := CleatControl = Cleat2And4;
END_IF;

(* Network 4 *)
_e4(CLK := CleatRollerSheetSense);
IF _e4.Q THEN
    blCleatFull := FALSE;
    blCleatFull := CleatControl = CleatFull;
END_IF;

(* Network 5 *)
cleat1 := (CEFNotchDetect OR cleat1) AND NOT CRReset AND NOT cleat4;

(* Network 6 *)
cleat2 := (NOT CEFNotchDetect OR cleat2) AND cleat1;

(* Network 7 *)
cleat3 := (CEFNotchDetect OR cleat3) AND cleat2;

(* Network 8 *)
cleat4 := NOT CEFNotchDetect AND cleat3;

(* Network 9 *)
CleatOutputRaw := (cleat1 AND ((NOT cleat2 AND blCleat1And3) OR blCleatFull)) OR (cleat3 AND NOT cleat4 AND blCleat2And4);

(* Network 10 *)
TON_0(IN := CleatOutputRaw, PT := tmCleatOnDelay);
CleatOutputDOM := TON_0.Q;

(* Network 11 *)
TOF_0(IN := CleatOutputDOM, PT := tmCleatOffDelay);
CleatOutputDOB := TOF_0.Q;

(* Network 12 *)
CleatOutput := CleatOutputDOM OR CleatOutputDOB;

(* Network 13 *)
LeftCleatKDRollValve := CleatOutput AND CleatLeft;

(* Network 14 *)
RightCleatKDRollValve := CleatOutput AND CleatRight;

(* Network 15 *)
TON_1(IN := cleat2 AND NOT cleat3, PT := T#2s);
CRReset := TON_1.Q;
END_PROGRAM
```

#### Init.ld
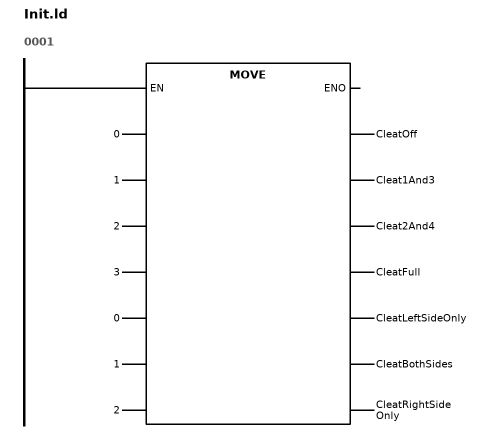
Ladder, written as Structured Text:
```iecst
PROGRAM _INIT
(* Network 1 *)
CleatOff := 0;
Cleat1And3 := 1;
Cleat2And4 := 2;
CleatFull := 3;
CleatLeftSideOnly := 0;
CleatBothSides := 1;
CleatRightSideOnly := 2;
END_PROGRAM
```

### Program Logical/SysCheck (IEC)

#### Cyclic.ld
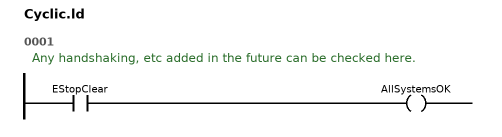
Ladder, written as Structured Text:
```iecst
PROGRAM _CYCLIC
(* Network 1: Any handshaking, etc added in the future can be checked here. *)
AllSystemsOK := EStopClear;
END_PROGRAM
```

#### Init.ld
Ladder, written as Structured Text:
```iecst
PROGRAM _INIT
(* Network 1 *)
END_PROGRAM
```

### Program Logical/SBrake (IEC)

#### Cyclic.ld - Cyclic code
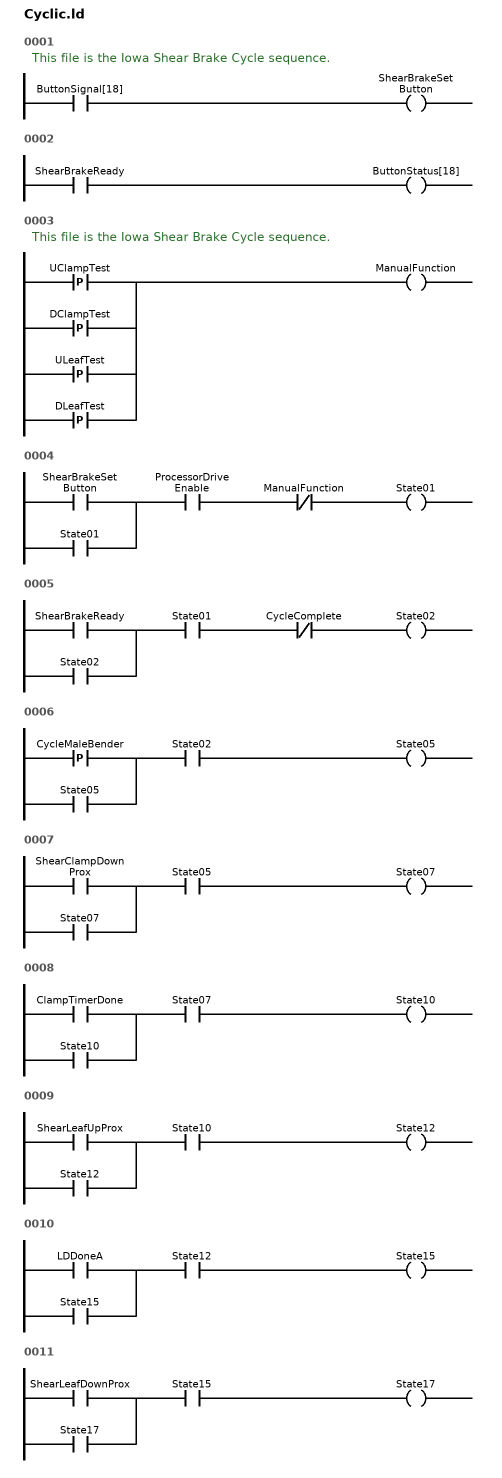
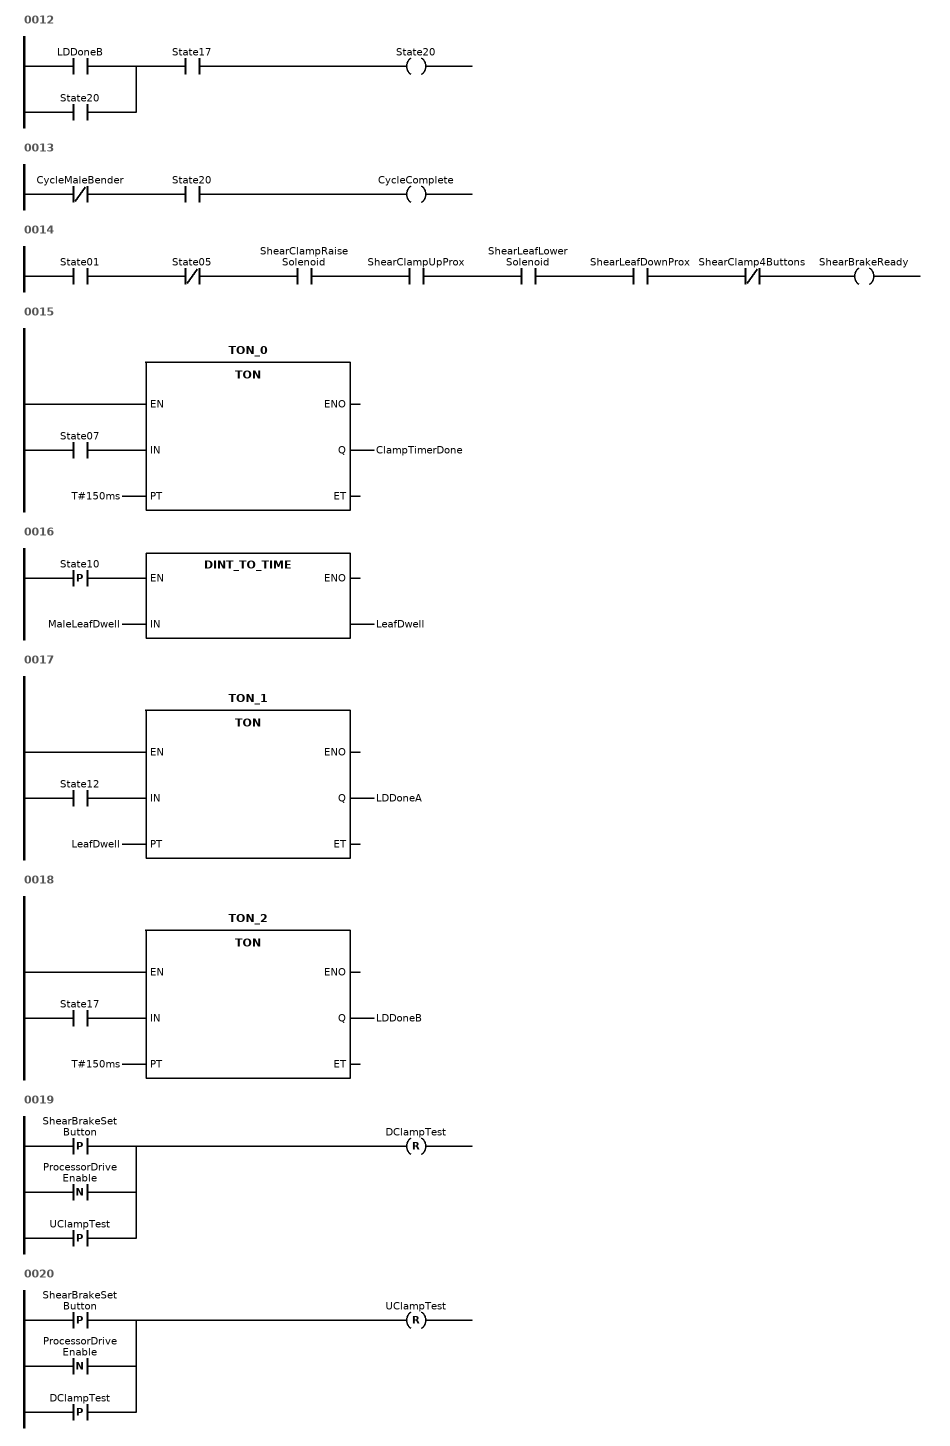
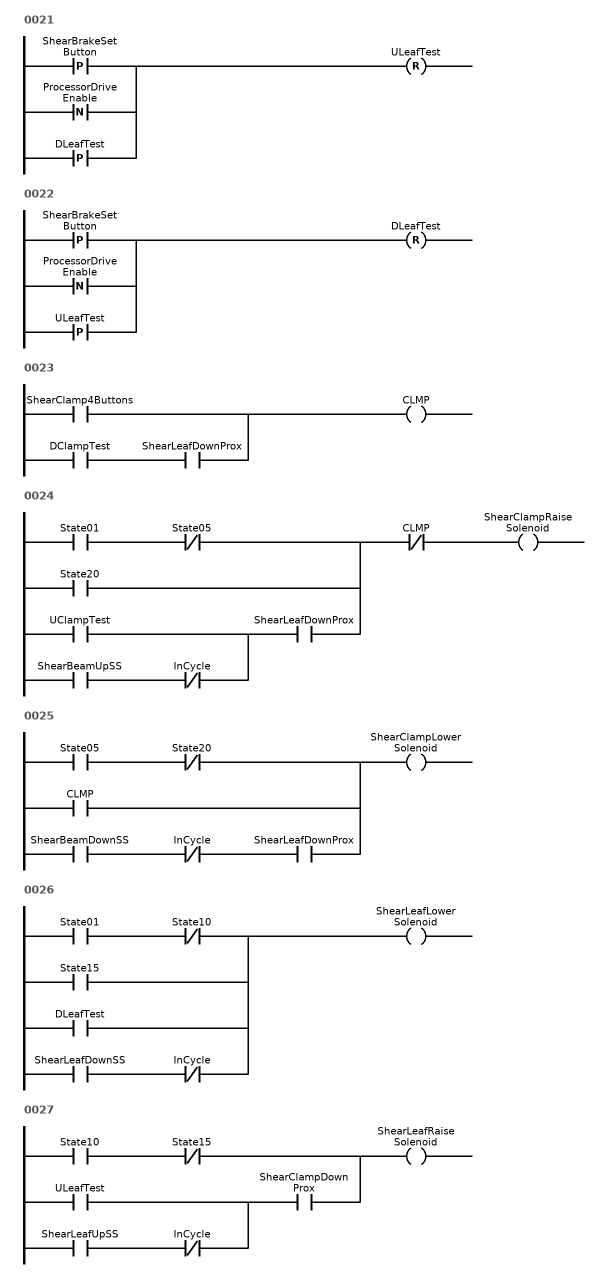
Ladder, written as Structured Text:
```iecst
PROGRAM _CYCLIC
VAR
    _e1 : R_TRIG;
    _e2 : R_TRIG;
    _e3 : R_TRIG;
    _e4 : R_TRIG;
    _e5 : R_TRIG;
    _e6 : R_TRIG;
    _e7 : R_TRIG;
    _e8 : F_TRIG;
    _e9 : R_TRIG;
    _e10 : R_TRIG;
    _e11 : F_TRIG;
    _e12 : R_TRIG;
    _e13 : R_TRIG;
    _e14 : F_TRIG;
    _e15 : R_TRIG;
    _e16 : R_TRIG;
    _e17 : F_TRIG;
    _e18 : R_TRIG;
END_VAR
(* Network 1: This file is the Iowa Shear Brake Cycle sequence. *)
ShearBrakeSetButton := ButtonSignal[18];

(* Network 2 *)
ButtonStatus[18] := ShearBrakeReady;

(* Network 3: This file is the Iowa Shear Brake Cycle sequence. *)
_e1(CLK := UClampTest);
_e2(CLK := DClampTest);
_e3(CLK := ULeafTest);
_e4(CLK := DLeafTest);
ManualFunction := _e1.Q OR _e2.Q OR _e3.Q OR _e4.Q;

(* Network 4 *)
State01 := (ShearBrakeSetButton OR State01) AND ProcessorDriveEnable AND NOT ManualFunction;

(* Network 5 *)
State02 := (ShearBrakeReady OR State02) AND State01 AND NOT CycleComplete;

(* Network 6 *)
_e5(CLK := CycleMaleBender);
State05 := (_e5.Q OR State05) AND State02;

(* Network 7 *)
State07 := (ShearClampDownProx OR State07) AND State05;

(* Network 8 *)
State10 := (ClampTimerDone OR State10) AND State07;

(* Network 9 *)
State12 := (ShearLeafUpProx OR State12) AND State10;

(* Network 10 *)
State15 := (LDDoneA OR State15) AND State12;

(* Network 11 *)
State17 := (ShearLeafDownProx OR State17) AND State15;

(* Network 12 *)
State20 := (LDDoneB OR State20) AND State17;

(* Network 13 *)
CycleComplete := NOT CycleMaleBender AND State20;

(* Network 14 *)
ShearBrakeReady := State01 AND NOT State05 AND ShearClampRaiseSolenoid AND ShearClampUpProx AND ShearLeafLowerSolenoid AND ShearLeafDownProx AND NOT ShearClamp4Buttons;

(* Network 15 *)
TON_0(IN := State07, PT := T#150ms);
ClampTimerDone := TON_0.Q;

(* Network 16 *)
_e6(CLK := State10);
IF _e6.Q THEN LeafDwell := DINT_TO_TIME(MaleLeafDwell); END_IF;

(* Network 17 *)
TON_1(IN := State12, PT := LeafDwell);
LDDoneA := TON_1.Q;

(* Network 18 *)
TON_2(IN := State17, PT := T#150ms);
LDDoneB := TON_2.Q;

(* Network 19 *)
_e7(CLK := ShearBrakeSetButton);
_e8(CLK := ProcessorDriveEnable);
_e9(CLK := UClampTest);
IF _e7.Q OR _e8.Q OR _e9.Q THEN DClampTest := FALSE; END_IF;

(* Network 20 *)
_e10(CLK := ShearBrakeSetButton);
_e11(CLK := ProcessorDriveEnable);
_e12(CLK := DClampTest);
IF _e10.Q OR _e11.Q OR _e12.Q THEN UClampTest := FALSE; END_IF;

(* Network 21 *)
_e13(CLK := ShearBrakeSetButton);
_e14(CLK := ProcessorDriveEnable);
_e15(CLK := DLeafTest);
IF _e13.Q OR _e14.Q OR _e15.Q THEN ULeafTest := FALSE; END_IF;

(* Network 22 *)
_e16(CLK := ShearBrakeSetButton);
_e17(CLK := ProcessorDriveEnable);
_e18(CLK := ULeafTest);
IF _e16.Q OR _e17.Q OR _e18.Q THEN DLeafTest := FALSE; END_IF;

(* Network 23 *)
CLMP := ShearClamp4Buttons OR (DClampTest AND ShearLeafDownProx);

(* Network 24 *)
ShearClampRaiseSolenoid := ((State01 AND NOT State05) OR State20 OR ((UClampTest OR (ShearBeamUpSS AND NOT InCycle)) AND ShearLeafDownProx)) AND NOT CLMP;

(* Network 25 *)
ShearClampLowerSolenoid := (State05 AND NOT State20) OR CLMP OR (ShearBeamDownSS AND NOT InCycle AND ShearLeafDownProx);

(* Network 26 *)
ShearLeafLowerSolenoid := (State01 AND NOT State10) OR State15 OR DLeafTest OR (ShearLeafDownSS AND NOT InCycle);

(* Network 27 *)
ShearLeafRaiseSolenoid := (State10 AND NOT State15) OR ((ULeafTest OR (ShearLeafUpSS AND NOT InCycle)) AND ShearClampDownProx);
END_PROGRAM
```

#### Variables.var - Local variables
```iecst
VAR
	State01 : BOOL;
	State02 : BOOL;
	State05 : BOOL;
	ManualFunction : BOOL;
	CycleComplete : BOOL;
	State07 : BOOL;
	TON_0 : TON;
	ClampTimerDone : BOOL;
	State10 : BOOL;
	State12 : BOOL;
	LDDoneA : BOOL;
	State15 : BOOL;
	State17 : BOOL;
	LDDoneB : BOOL;
	State20 : BOOL;
	LeafDwell : TIME;
	TON_1 : TON;
	TON_2 : TON;
	CLMP : BOOL;
END_VAR
```

### Program Logical/EFeeder1 (IEC)

#### Variables.var
```iecst
VAR
	AnalogForward : BOOL;
	AnalogReverse : BOOL;
	AutoSignal : BOOL;
	BatchCancelUnlatch : BOOL;
	BeadRollFires : BOOL;
	BeadRollUsedUp : BOOL;
	Block_1 : BOOL;
	ButtonBack7 : BOOL;
	ButtonFires : BOOL;
	ButtonUsedUp : BOOL;
	CenterHoleFires : BOOL;
	CenterHoleTime : TIME;
	CenterHoleUsedUp : BOOL;
	CenterPosA : BOOL;
	CenterShuttleIndex : INT;
	ChangeCShuttle : BOOL;
	ChangeJob1 : BOOL;
	ChangeLShuttle : BOOL;
	ChangeRShuttle : BOOL;
	ClearEncoderSignal : BOOL;
	CleatFires : BOOL;
	CleatUsedUp : BOOL;
	CLPUnlatch : BOOL;
	CShuttleUnlatch : BOOL;
	CustomLTFires : BOOL;
	CustomLTTime : TIME;
	CustomLTUsedUp : BOOL;
	CustomLTValve : BOOL;
	CustomVFires : BOOL;
	CustomVTime : TIME;
	CustomVUsedUp : BOOL;
	DamperLatch : BOOL;
	DamperResult : DINT;
	DataUpdated : BOOL;
	DDDoneTimer : TON;
	DieDelayDone : BOOL;
	DieUpTime : TIME;
	DirectionDelayDone : BOOL;
	DuctoAutoUnlatch : BOOL;
	FFCLatch : BOOL;
	FiveFootCoil : BOOL;
	FourFootCoil : BOOL;
	FourResult : DINT;
	GapPulse : BOOL;
	GapTP : BOOL;
	GTime : TIME;
	HalfUpdated1 : BOOL;
	HalfUpdated2 : BOOL;
	HolePunchSelecedtSolenoid : BOOL;
	IncPartsMade : BOOL;
	InitMoveSignal : BOOL;
	InPositionBand : REAL := 0.01;
	JobChanging : BOOL;
	LeftHoleFires : BOOL;
	LeftHoleTime : TIME;
	LeftHoleUsedUp : BOOL;
	LeftPosA : BOOL;
	LTFires : BOOL;
	LTTime : TIME;
	LTUsedUp : BOOL;
	ManualSignal : BOOL;
	MarkAccumulator : REAL;
	MetalEncoderLatch : DINT;
	NewRunJobOk : BOOL;
	NextMoveComplete : BOOL;
	NextMoveLookAgain : BOOL;
	NoShearHits : BOOL;
	OGLatch : BOOL;
	OGResult : DINT;
	OneResult : DINT;
	OutsideLatch : BOOL;
	PartCutOff : BOOL;
	PartRefOK : BOOL;
	PunchCurrentSelect : DINT;
	RightHoleFires : BOOL;
	RightHoleTime : TIME;
	RightHoleUsedUp : BOOL;
	RightPosA : BOOL;
	RollEnableUnlatch : BOOL;
	RShuttleUnlatch : BOOL;
	RTotalInches : REAL;
	RunSpeedCalculated : BOOL;
	SetConnectorChange : BOOL;
	ShearBrakeFires : BOOL;
	ShearBrakeUsedUp : BOOL;
	ShearFires : BOOL;
	ShearHitsLTZero : BOOL;
	shearTime : TIME;
	ShearUsedUp : BOOL;
	SixFootCoil : BOOL;
	SmallResult : REAL;
	Step04A : BOOL;
	Step05A : BOOL;
	Step05B : BOOL;
	Step06 : BOOL;
	Step07 : BOOL;
	Step08 : BOOL;
	Step09 : BOOL;
	Step10 : BOOL;
	Step15 : BOOL;
	Step16 : BOOL;
	Step17 : BOOL;
	Step18 : BOOL;
	Step18A : BOOL;
	Step18B : BOOL;
	Step19 : BOOL;
	ThirdOff1 : BOOL;
	ThirdOff2 : BOOL;
	ThirdOff3 : BOOL;
	TON_0 : TON;
	TON_1 : TON;
	TON_10 : TON;
	TON_Warning : TON;
	TP_0 : TP;
	TP_1 : TP;
	TP_2 : TP;
	TP_3 : TP;
	TP_4 : TP;
	TP_5 : TP;
	TP_6 : TP;
	TP_7 : TP;
	TP_8 : TP;
	TP_9 : TP;
	UnlatchBender : BOOL;
	UnlatchButtons : BOOL;
	VFires : BOOL;
	VTime : TIME;
	VUsedUp : BOOL;
	Wait1Ready : BOOL;
	Wait2Ready : BOOL;
	Wait3Ready : BOOL;
	WaitCon1 : BOOL;
	WaitCon2 : BOOL;
	ZCOLT0 : BOOL;
	ZCReverseComplete : BOOL;
	ZCSCTimer : TON;
	ZCSettleComplete : BOOL;
	ZeroCropDifference : DINT;
	ZRCTon : TON;
	FinalScan : BOOL;
	Step12 : BOOL;
	SHLT0 : BOOL;
	Step20 : BOOL;
	ReturnTarget : DINT;
	ReturnComplete : BOOL;
	Step21 : BOOL;
	ReturnCalculated : BOOL;
	Step22 : BOOL;
	JobsDifferent : BOOL;
END_VAR
```

#### Action.st
```iecst
ACTION myAction:
	IF ShearHits < 120000 THEN
		ShearHits := ShearHits + 1;
	END_IF;

END_ACTION

ACTION getNextMove:
	(*Find smallest move*)
	(*The shear will always be used*)
	IF getNextMove.x AND NOT getNextMove._x THEN
		FinalScan := TRUE;
	ELSE
		NextMoveDone := TRUE;
		SmallResult := ShearMove;
		IF LTNotchMove < SmallResult AND LTNotchMove > InvalidDistREAL THEN
			SmallResult := LTNotchMove;
		END_IF;
		IF VNotchMove < SmallResult AND VNotchMove > InvalidDistREAL THEN
			SmallResult := VNotchMove;
		END_IF;
		IF LeftHoleMove < SmallResult AND LeftHoleMove > InvalidDistREAL THEN
			SmallResult := LeftHoleMove;
		END_IF;
		IF CenterHoleMove < SmallResult AND CenterHoleMove > InvalidDistREAL THEN
			SmallResult := CenterHoleMove;
		END_IF;
		IF RightHoleMove < SmallResult AND RightHoleMove > InvalidDistREAL THEN
			SmallResult := RightHoleMove;
		END_IF;
		IF ButtonMove < SmallResult AND ButtonMove > InvalidDistREAL THEN
			SmallResult := ButtonMove;
		END_IF;
		IF ShearBrakeMove < SmallResult AND ShearBrakeMove > InvalidDistREAL THEN
			SmallResult := ShearBrakeMove;
		END_IF;
		IF CustomLTMove < SmallResult AND CustomLTMove > InvalidDistREAL THEN
			SmallResult := CustomLTMove;
		END_IF;
		IF CleatMove < SmallResult AND CleatMove > InvalidDistREAL THEN
			SmallResult := CleatMove;
		END_IF;
		IF CustomVMove < SmallResult AND CustomVMove > InvalidDistREAL THEN
			SmallResult := CustomVMove;
		END_IF;
		(*IF BeadRollMove < SmallResult AND BeadRollMove > InvalidDistREAL THEN
			SmallResult := BeadRollMove;
		END_IF;*)

		ShearMove := ShearMove - SmallResult;
		IF LTNotchMove > InvalidDistREAL THEN
			LTNotchMove := LTNotchMove - SmallResult;
		END_IF;
		IF VNotchMove > InvalidDistREAL THEN
			VNotchMove := VNotchMove - SmallResult;
		END_IF;
		IF LeftHoleMove > InvalidDistREAL THEN
			LeftHoleMove := LeftHoleMove - SmallResult;
		END_IF;
		IF CenterHoleMove > InvalidDistREAL THEN
			CenterHoleMove := CenterHoleMove - SmallResult;
		END_IF;
		IF RightHoleMove > InvalidDistREAL THEN
			RightHoleMove := RightHoleMove - SmallResult;
		END_IF;
		IF ButtonMove > InvalidDistREAL THEN
			ButtonMove := ButtonMove - SmallResult;
		END_IF;
		IF ShearBrakeMove > InvalidDistREAL THEN
			ShearBrakeMove := ShearBrakeMove - SmallResult;
		END_IF;
		IF CustomLTMove > InvalidDistREAL THEN
			CustomLTMove := CustomLTMove - SmallResult;
		END_IF;
		IF CleatMove > InvalidDistREAL THEN
			CleatMove := CleatMove - SmallResult;
		END_IF;
		IF CustomVMove > InvalidDistREAL THEN
			CustomVMove := CustomVMove - SmallResult;
		END_IF;
		(*IF BeadRollMove > InvalidDistREAL THEN
			BeadRollMove := BeadRollMove - SmallResult;
		END_IF;*)
	END_IF;
END_ACTION

ACTION UpdateTables:
	IF UpdateTables.x AND NOT UpdateTables._x THEN
		FinalScan := TRUE;
	ELSE
		UpdateTablesDone := TRUE;
		IF ShearUsedUp AND ShearHits > 0 THEN
			ShearFires := TRUE;
			ShearHits := ShearHits - 1;
			(*Do this before the index changes *)
			IF (ShearIndex = 0 AND ShearFFlag = 1) OR
				(ShearIndex = 1 AND ShearTable[2] <= InvalidDistREAL) OR
				(ShearIndex = 2) THEN
				PartCutOff := TRUE;
			END_IF;
			ShearIndex := ShearIndex + 1;
			IF ShearTable[ShearIndex] <= InvalidDistREAL THEN
				ShearIndex := 1;
			END_IF;
			IF ShearHits <= 0 THEN
				MakeShearTable := TRUE;
				ShearIndex := 0;
			END_IF;
		END_IF;
		IF LTUsedUp THEN
			IF LTNotchHits > 0 THEN
				LTFires := TRUE;
				LTNotchHits := LTNotchHits - 1;
			END_IF;
			LTNotchIndex := LTNotchIndex + 1;
			IF LTNotchTable[LTNotchIndex] <= InvalidDistREAL THEN
				LTNotchIndex := 1;
			END_IF;
			SavedConnector := LatestConnector;
			IF LTNotchHits <= 0 THEN
				MakeLTTable := TRUE;
				LTNotchIndex := 0;
			END_IF;
		END_IF;
		IF VUsedUp THEN
			IF VNotchHits > 0 THEN
				VFires := TRUE;
				VNotchHits := VNotchHits - 1;
			END_IF;
			VNotchIndex := VNotchIndex + 1;
			IF VNotchTable[VNotchIndex] <= InvalidDistREAL THEN
				VNotchIndex := 1;
			END_IF;
			IF VNotchHits <= 0 THEN
				MakeVTable := TRUE;
				VNotchIndex := 0;
			END_IF;
		END_IF;
		IF LeftHoleUsedUp THEN
			IF LeftHoleHits > 0 THEN
				LeftHoleFires := TRUE;
				LeftHoleHits := LeftHoleHits - 1;
			END_IF;
			LeftHoleIndex := LeftHoleIndex + 1;
			IF LeftHoleTable[LeftHoleIndex] <= InvalidDistREAL THEN
				LeftHoleIndex := 1;
			END_IF;
			IF LeftHoleHits <= 0 THEN
				MakeLHoleTable := TRUE;
				LeftHoleIndex := 0;
			END_IF;
		END_IF;
		IF CenterHoleUsedUp THEN
			IF CenterHoleHits > 0 THEN
				CenterHoleFires := TRUE;
				CenterHoleHits := CenterHoleHits - 1;
			END_IF;
			CenterHoleIndex := CenterHoleIndex + 1;
			IF CenterHoleTable[CenterHoleIndex] <= InvalidDistREAL THEN
				CenterHoleIndex := 1;
			END_IF;
			IF CenterHoleHits <= 0 THEN
				MakeCHoleTable := TRUE;
				CenterHoleIndex := 0;
			END_IF;
		END_IF;
		IF RightHoleUsedUp THEN
			IF RightHoleHits > 0 THEN
				RightHoleFires := TRUE;
				RightHoleHits := RightHoleHits - 1;
			END_IF;
			RightHoleIndex := RightHoleIndex + 1;
			IF RightHoleTable[RightHoleIndex] <= InvalidDistREAL THEN
				RightHoleIndex := 1;
			END_IF;
			IF RightHoleHits <= 0 THEN
				MakeRHoleTable := TRUE;
				RightHoleIndex := 0;
			END_IF;
		END_IF
		IF ButtonUsedUp THEN
			IF ButtonHits > 0 THEN
				ButtonFires := TRUE;
				ButtonHits := ButtonHits - 1;
			END_IF;
			ButtonIndex := ButtonIndex + 1;
			IF ButtonTable[ButtonIndex] <= InvalidDistREAL THEN
				ButtonIndex := 1;
			END_IF;
			IF ButtonHits <= 0 THEN
				MakeButtonTable := TRUE;
				ButtonIndex := 0;
			END_IF;
		END_IF;
		IF ShearBrakeUsedUp THEN
			IF ShearBrakeHits > 0 THEN
				ShearBrakeFires := TRUE;
				ShearBrakeHits := ShearBrakeHits - 1;
			END_IF;
			ShearBrakeIndex := ShearBrakeIndex + 1;
			IF ShearBrakeTable[ShearBrakeIndex] <= InvalidDistREAL THEN
				ShearBrakeIndex := 1;
			END_IF;
			IF ShearBrakeHits <= 0 THEN
				MakeShearBrakeTable := TRUE;
				ShearBrakeIndex := 0;
			END_IF;
		END_IF;
		IF CustomLTUsedUp THEN
			IF CustomLTHits > 0 THEN
				CustomLTFires := TRUE;
				CustomLTHits := CustomLTHits - 1;
			END_IF;
			CustomLTIndex := CustomLTIndex + 1;
			IF CustomLTTable[CustomLTIndex] <= InvalidDistREAL THEN
				CustomLTIndex := 1;
			END_IF;
			IF CustomLTHits <= 0 THEN
				MakeCustomLTTable := TRUE;
				CustomLTIndex := 0;
			END_IF;
		END_IF;
		IF CleatUsedUp THEN
			IF CleatHits > 0 THEN
				CleatFires := TRUE;
				CleatHits := CleatHits - 1;
			END_IF;
			CleatIndex := CleatIndex + 1;
			IF CleatTable[CleatIndex] <= InvalidDistREAL THEN
				CleatIndex := 1;
			END_IF;
			IF CleatHits <= 0 THEN
				MakeCleatTable := TRUE;
				CleatIndex := 0;
			END_IF;
		END_IF;
		IF CustomVUsedUp THEN
			IF CustomVHits > 0 THEN
				CustomVFires := TRUE;
				CustomVHits := CustomVHits - 1;
			END_IF;
			CustomVIndex := CustomVIndex + 1;
			IF CustomVTable[CustomVIndex] <= InvalidDistREAL THEN
				CustomVIndex := 1;
			END_IF;
			IF CustomVHits <= 0 THEN
				MakeCustomVTable := TRUE;
				CustomVIndex := 0;
			END_IF;
		END_IF;
		(*IF BeadRollUsedUp THEN
			IF BeadRollHits > 0 THEN
				BeadRollFires := TRUE;
				BeadRollHits := BeadRollHits - 1;
			END_IF;
			BeadRollIndex := BeadRollIndex + 1;
			IF BeadRollTable[BeadRollIndex] <= InvalidDistREAL THEN
				BeadRollIndex := 1;
			END_IF;
			IF BeadRollHits <= 0 THEN
				MakeBeadRollTable := TRUE;
				BeadRollIndex := 0;
			END_IF;
		END_IF; *)
	END_IF;
END_ACTION
```
